FUNCTION_BLOCK ABSTRACT FB_String_Enumerator_Base IMPLEMENTS I_Enumerator
VAR
	Index : T_Size := -1;
END_VAR

(* Gets current string representation of element*)
PROPERTY ABSTRACT _Current : T_Long_String
GET
END_GET
END_PROPERTY

(* Gets current element. Returns TRUE if retrieval and converstion was successful.*)
METHOD ABSTRACT Current : BOOL
VAR_INPUT
	sValue : REFERENCE TO STRING;
END_VAR
END_METHOD

(* Disposes or release resources for specified task*)
METHOD Dispose
END_METHOD

(* Advances enumerator to the next element. On first call or after reset it generates new element data to enumerate over.*)
METHOD ABSTRACT Next : BOOL
END_METHOD

(* Sets enumerator to it's intial position. Disposes data pertaining to it's old elements.*)
METHOD Reset
THIS^.Index := -1;
END_METHOD

END_FUNCTION_BLOCK

(* stored: Version 1.1.0.1, ProductVersion 3.1.4024.4
   POU FB_String_Enumerator_Base: Id {53f5a01b-897d-4fc6-a5cb-1e89395b8ce3}, SpecialFunc None
   Property _Current: Id {e14637df-31b7-4c65-bc62-5176a363a474}
   Get Get: Id {7bcd9739-d388-46f6-b2f3-c3da901815ba}
   Method Current: Id {82173c8e-1dca-4189-aa46-53fee7e0a36e}
   Method Dispose: Id {95ab4e17-76c0-4363-a0e2-ad9634c110b6}
   Method Next: Id {5eca136a-40e5-4f5e-baa2-f6eb76c7383f}
   Method Reset: Id {55d0860d-ce83-4e49-9272-08ee65cd9b58} *)
